// TIA Portal V19 export
TYPE "TAx_DriveInterface"
// stored: Access Published
   STRUCT
      Infeed_ON : Bool;   // Infeed running (enabled)
      AccessPoint : HW_IO;   // AccesPoint for SinaParaS
      AxisID : USInt;   // Axis ID for SinaParaS
      TokenChain : Int;   // Number of token chain for SinaParaS
   END_STRUCT;
END_TYPE
